// TIA Portal V18 export
DATA_BLOCK "TD_Start_Elec_DB"   // DB13
// stored: AutoNumber false, InstanceOfName TD_Motor_Start_Elec, InstanceOfType FB
"TD_Motor_Start_Elec"
   // VAR
   //    TDP1FailTON { S7_SetPoint := 'True'} : TON_TIME;
   //    TDP2FailTON { S7_SetPoint := 'True'} : TON_TIME;
   // END_VAR
BEGIN
END_DATA_BLOCK
